Staubli VAL3: moveManager.pgx

program moveManager(joint destination (dimensions=1), mdesc armSpeed (dimensions=1), string reply (dimensions=1), num sio_ID (dimensions=1))
begin
  //**************************************************
  // Method to enable joint-based movements of the robot. The referenced
  // observeStop() method allows interrupts/restarts to be handled
  //**************************************************
  moveIsStopped=false
  taskCreate "observeStop",5,observeStop()
  movej(destination,flange,armSpeed)
  waitEndMove()
  taskCreate "sendStatus",10,sendStatus(reply,sio_ID)
  taskKill("observeStop")
end
